PROGRAM P_Demo_PUDINT_TO_UDINT
VAR
    nRealValue           : UDINT := 4000000000; // 模拟 wire 缓冲区中的 UDINT 字段
    pUDINTField          : POINTER TO UDINT; // 业务侧先算好的字段地址（ADR 或 pBase+nOff）
    bExtractField        : BOOL; // 在线置 TRUE 触发一次解析
    nRealValue_extracted : UDINT; // 解析后的副本，供业务逻辑使用
END_VAR

// ============================================================
// Tc2_Utilities.PUDINT_TO_UDINT 演示程序（FUNCTION）
// ============================================================
// 场景：从一段二进制 wire 缓冲区里按偏移取 UDINT 字段（Modbus/CAN/ADS Raw）。
// 价值：替代手写 pField + nOff + ^ 指针算术；一次调用取值，少打错符号。
// 验证：在线写 nRealValue := 4000000000；bExtractField := TRUE；
//       下一周期 nRealValue_extracted 应等于 nRealValue。
// ============================================================

// 业务代码通常已经算好字段地址（pBase + 协议偏移）；演示用 ADR 等价
pUDINTField := ADR(nRealValue);

IF bExtractField AND pUDINTField <> 0 THEN
    // 单次完整调用：避免手写 ^ 解引用，统一风格便于和字节序转换串联
    nRealValue_extracted := PUDINT_TO_UDINT(pUDINTField);
    bExtractField := FALSE;
END_IF;

END_PROGRAM

(* stored: Version 1.1.0.1, ProductVersion 3.1.4024.5
   POU P_Demo_PUDINT_TO_UDINT: Id {56b0df90-a07d-59fe-9517-5c11826f9857}, SpecialFunc None *)
